FUNCTION_BLOCK RunBin EXTENDS RunUnitGeneric
VAR_INPUT
	sensor : POINTER TO RunSignal;
END_VAR
VAR_OUTPUT
	collectionCount AT%M*: UDINT;
END_VAR
VAR
	ready AT%Q* : BOOL;
	ack AT%I* : BOOL;
	
	tickTime AT%Q*: DWORD ; //in ms
	
	totalCount AT%M* : UDINT; //wonld't be reset for each batch
END_VAR
VAR PERSISTENT
	collectionLimit AT%M* : UINT;
END_VAR

SUPER^();


CASE outputState OF
	eSpecialStates.INITIAL_BEGIN:
		collectionCount := 0;
		NextState := eSpecialStates.INITIAL_END;
	//-----------------
	//	START
	//-----------------
	eSpecialStates.GENERIC_GROUP_START:
		bSerialTransition := (collectionCount < collectionLimit) AND  (sensor <> 0 AND_THEN sensor^.debouncedOn);
		IF bSerialTransition THEN
			ready := TRUE;
			workingTimer.IN := TRUE; //start counting
		ELSIF collectionCount <> 0 AND (sensor <> 0 AND_THEN NOT sensor^.debouncedOn) THEN
			collectionCount := 0; //count reset
		END_IF
	1:
		bSerialTransition := ack;
		IF bSerialTransition THEN
			
			//tick time calculation
			tickTime := TIME_TO_DWORD(workingTimer.ET);
			workingTimer.IN := FALSE;
		
			collectionCount := IncNoOverflow(input:= collectionCount);
			totalCount := IncNoOverflow(input:= totalCount);
			
			ready := FALSE;
		ELSIF sensor <> 0 AND_THEN NOT sensor^.debouncedOn THEN
			ready := FALSE;
			NextState := 0; //re=scan
		END_IF
	2: 
		bSerialTransition := NOT ack;
		IF bSerialTransition THEN
			NextState := eSpecialStates.GENERIC_GROUP_START;
		END_IF
END_CASE

END_FUNCTION_BLOCK

(* stored: Version 1.1.0.1, ProductVersion 3.1.4024.0
   POU RunBin: Id {0bf50b34-1c3e-4db6-842a-bc6f0d7033ed}, SpecialFunc None *)
